PROGRAM MAIN
VAR
    // ── Per-valve motion controllers ──────────────────────────
    fbValve1 : FB_ValveControl;
    fbValve2 : FB_ValveControl;
    fbValve3 : FB_ValveControl;

    // ── NC axis references (linked in TwinCAT I/O mapping) ───
    Axis_Valve1 : AXIS_REF;
    Axis_Valve2 : AXIS_REF;
    Axis_Valve3 : AXIS_REF;

    // ── Infrastructure function blocks ────────────────────────
    fbCsvLogger   : FB_CsvLogger;
    fbMqttManager : FB_MqttManager;

    // ── Internal buffers for MQTT status publishing ───────────
    arrValveSetpoint : ARRAY[1..3] OF REAL;
    arrValveActual   : ARRAY[1..3] OF REAL;
    arrValveSource   : ARRAY[1..3] OF STRING(32);

    // ── Internal helpers ──────────────────────────────────────
    arrPrevHmiSetpoint : ARRAY[1..3] OF REAL := [-1.0, -1.0, -1.0];
    iValve : INT;
END_VAR

// ============================================================
// MAIN PROGRAM OVERVIEW (NOVICE GUIDE)
// ------------------------------------------------------------
// This program is the "orchestrator" of the whole irrigation PLC:
// - It reads operator requests from HMI.
// - It reads remote requests from MQTT (if enabled by operator).
// - It decides which source currently controls each valve.
// - It calls each valve motion FB once per PLC cycle.
// - It logs process values to CSV and mirrors status back to HMI.
//
// Execution sequence each PLC cycle:
// 1) Read/limit HMI commands and reset commands
// 2) Handle source arbitration (HMI vs MQTT)
// 3) Run valve FBs (motion execution)
// 4) Run CSV logger
// 5) Update HMI feedback + overall system health flags
// ============================================================

// ------------------------------------------------------------
// 1) Read and sanitize HMI commands
// ------------------------------------------------------------
GVL_System.Valve[1].HMI_Setpoint := LIMIT(0.0, GVL_HMI.HMI_Valve1_Setpoint, 100.0);
GVL_System.Valve[2].HMI_Setpoint := LIMIT(0.0, GVL_HMI.HMI_Valve2_Setpoint, 100.0);
GVL_System.Valve[3].HMI_Setpoint := LIMIT(0.0, GVL_HMI.HMI_Valve3_Setpoint, 100.0);

GVL_System.Valve[1].Reset_Cmd := GVL_HMI.HMI_Valve1_Reset;
GVL_System.Valve[2].Reset_Cmd := GVL_HMI.HMI_Valve2_Reset;
GVL_System.Valve[3].Reset_Cmd := GVL_HMI.HMI_Valve3_Reset;

IF GVL_HMI.HMI_ResetAll THEN
    GVL_System.Valve[1].Reset_Cmd := TRUE;
    GVL_System.Valve[2].Reset_Cmd := TRUE;
    GVL_System.Valve[3].Reset_Cmd := TRUE;
    GVL_HMI.HMI_ResetAll := FALSE;
END_IF

// ------------------------------------------------------------
// 2) HMI/MQTT command source handling
// ------------------------------------------------------------
// Arbitration rule for beginners:
// - By default, first valid source is HMI.
// - If operator changes HMI setpoint, active source becomes HMI.
// - If a new valid MQTT command arrives and MQTT is enabled,
//   active source changes to MQTT for that valve.
// - Source is stored in GVL_System.Valve[i].Source and shown on HMI.
FOR iValve := 1 TO 3 DO
    IF GVL_System.Valve[iValve].Source = E_ValveSource.NONE THEN
        GVL_System.Valve[iValve].Source := E_ValveSource.HMI;
        GVL_System.Valve[iValve].Active_Setpoint := GVL_System.Valve[iValve].HMI_Setpoint;
    END_IF

    IF ABS(GVL_System.Valve[iValve].HMI_Setpoint - arrPrevHmiSetpoint[iValve]) > 0.001 THEN
        GVL_System.Valve[iValve].Active_Setpoint := GVL_System.Valve[iValve].HMI_Setpoint;
        GVL_System.Valve[iValve].Source := E_ValveSource.HMI;
        arrPrevHmiSetpoint[iValve] := GVL_System.Valve[iValve].HMI_Setpoint;
    END_IF
END_FOR

// Prepare status arrays before MQTT publish
// (This is done in arrays because FB_MqttManager expects fixed arrays.)
arrValveSetpoint[1] := GVL_System.Valve[1].Active_Setpoint;
arrValveSetpoint[2] := GVL_System.Valve[2].Active_Setpoint;
arrValveSetpoint[3] := GVL_System.Valve[3].Active_Setpoint;
arrValveActual[1] := GVL_System.Valve[1].Actual_Position;
arrValveActual[2] := GVL_System.Valve[2].Actual_Position;
arrValveActual[3] := GVL_System.Valve[3].Actual_Position;
arrValveSource[1] := TO_STRING(GVL_System.Valve[1].Source);
arrValveSource[2] := TO_STRING(GVL_System.Valve[2].Source);
arrValveSource[3] := TO_STRING(GVL_System.Valve[3].Source);

// MQTT enable is operator-controlled from HMI checkbox.
// Broker/topic/timing configuration stays fixed in code constants
// (single source of truth = GVL_Config.MQTT_CONFIG).
fbMqttManager(
    bEnable              := GVL_HMI.HMI_MQTT_bEnable,
    stConfig             := GVL_Config.MQTT_CONFIG,
    bApplyConfig         := FALSE,
    bPublish             := GVL_HMI.HMI_MQTT_mPublish,
    sPubTopic            := GVL_Config.MQTT_CONFIG.sMainTopic,
    sPubPayload          := '',
    bSubscribe           := GVL_HMI.HMI_MQTT_bEnable,
    sSubTopic            := GVL_Config.MQTT_CONFIG.SubscribeTopic,
    bUnsubscribe         := FALSE,
    sUnsubTopic          := '',
    bEnableStatusPublish := GVL_HMI.HMI_MQTT_bEnable,
    tStatusPublishTime   := GVL_Config.MQTT_CONFIG.tPublishInterval,
    sStatusTopic         := GVL_Config.MQTT_CONFIG.sMainTopic,
    rValveSetpoint       := arrValveSetpoint,
    rValveActual         := arrValveActual,
    sValveSource         := arrValveSource,
    rTemperature_C       := INT_TO_REAL(GVL_IO.AI_Tmp_1),
    rWaterLevel_Percent  := INT_TO_REAL(GVL_IO.AI_L1V11),
    sTimestamp           := DT_TO_STRING(CURRENT_DT())
);

IF fbMqttManager.bNewRemoteCommand AND GVL_HMI.HMI_MQTT_bEnable THEN
    FOR iValve := 1 TO 3 DO
        GVL_System.Valve[iValve].MQTT_Setpoint   := fbMqttManager.rMqttValveSetpoint[iValve];
        GVL_System.Valve[iValve].Active_Setpoint := GVL_System.Valve[iValve].MQTT_Setpoint;
        GVL_System.Valve[iValve].Source          := E_ValveSource.MQTT;
    END_FOR
END_IF

// ------------------------------------------------------------
// 3) Valve motion control calls (one FB per valve axis)
// Each FB handles homing, move, halt, reset, and fault state machine
// for its own NC axis. MAIN only forwards commands/parameters.
// ------------------------------------------------------------
fbValve1(
    Axis            := Axis_Valve1,
    HMI_Setpoint    := GVL_System.Valve[1].HMI_Setpoint,
    MQTT_Setpoint   := GVL_System.Valve[1].MQTT_Setpoint,
    MQTT_Enabled    := GVL_HMI.HMI_MQTT_bEnable,
    Enable          := TRUE,
    eHomingSelection:= MC_Direct,
    Reset           := GVL_System.Valve[1].Reset_Cmd,
    MoveVelocity    := GVL_Config.VALVE_MOVE_VELOCITY,
    MoveAccel       := GVL_Config.VALVE_MOVE_ACCELERATION,
    MoveDecel       := GVL_Config.VALVE_MOVE_DECELERATION,
    MoveJerk        := GVL_Config.VALVE_MOVE_JERK,
    HomeVelocity    := GVL_Config.VALVE_HOMING_VELOCITY,
    FullStroke_mm   := GVL_Config.VALVE_FULL_STROKE_MM,
    PosTolerance    := GVL_Config.VALVE_POSITION_TOLERANCE,
    Move_Stop       := GVL_HMI.HMI_Valve1_Stop,
    UPDATE          := GVL_HMI.HMI_UPDATE,
    ZeroPosition    := GVL_IO.bBottom_position_1,
    bHoming         := GVL_HMI.HMI_Valve1_Homing,
    Actual_Position => GVL_System.Valve[1].Actual_Position,
    State           => GVL_System.Valve[1].State,
    Source          => GVL_System.Valve[1].Source,
    IsHomed         => GVL_System.Valve[1].IsHomed,
    InPosition      => GVL_System.Valve[1].InPosition,
    IsFault         => GVL_System.Valve[1].IsFault,
    FaultCode       => GVL_System.Valve[1].FaultCode,
    rTarget_mm      => GVL_HMI.Raw_Valve1_Setpoint,
    rActual_mm      => GVL_HMI.Raw_Valve1_Position
);

fbValve2(
    Axis            := Axis_Valve2,
    HMI_Setpoint    := GVL_System.Valve[2].HMI_Setpoint,
    MQTT_Setpoint   := GVL_System.Valve[2].MQTT_Setpoint,
    MQTT_Enabled    := GVL_HMI.HMI_MQTT_bEnable,
    Enable          := TRUE,
    eHomingSelection:= MC_Direct,
    Reset           := GVL_System.Valve[2].Reset_Cmd,
    MoveVelocity    := GVL_Config.VALVE_MOVE_VELOCITY,
    MoveAccel       := GVL_Config.VALVE_MOVE_ACCELERATION,
    MoveDecel       := GVL_Config.VALVE_MOVE_DECELERATION,
    MoveJerk        := GVL_Config.VALVE_MOVE_JERK,
    HomeVelocity    := GVL_Config.VALVE_HOMING_VELOCITY,
    FullStroke_mm   := GVL_Config.VALVE_FULL_STROKE_MM,
    PosTolerance    := GVL_Config.VALVE_POSITION_TOLERANCE,
    Move_Stop       := GVL_HMI.HMI_Valve2_Stop,
    UPDATE          := GVL_HMI.HMI_UPDATE,
    bHoming         := GVL_HMI.HMI_Valve2_Homing,
    Actual_Position => GVL_System.Valve[2].Actual_Position,
    State           => GVL_System.Valve[2].State,
    Source          => GVL_System.Valve[2].Source,
    IsHomed         => GVL_System.Valve[2].IsHomed,
    InPosition      => GVL_System.Valve[2].InPosition,
    IsFault         => GVL_System.Valve[2].IsFault,
    FaultCode       => GVL_System.Valve[2].FaultCode,
    rTarget_mm      => GVL_HMI.Raw_Valve2_Setpoint,
    rActual_mm      => GVL_HMI.Raw_Valve2_Position
);

fbValve3(
    Axis            := Axis_Valve3,
    HMI_Setpoint    := GVL_System.Valve[3].HMI_Setpoint,
    MQTT_Setpoint   := GVL_System.Valve[3].MQTT_Setpoint,
    MQTT_Enabled    := GVL_HMI.HMI_MQTT_bEnable,
    Enable          := TRUE,
    eHomingSelection:= MC_Direct,
    Reset           := GVL_System.Valve[3].Reset_Cmd,
    MoveVelocity    := GVL_Config.VALVE_MOVE_VELOCITY,
    MoveAccel       := GVL_Config.VALVE_MOVE_ACCELERATION,
    MoveDecel       := GVL_Config.VALVE_MOVE_DECELERATION,
    MoveJerk        := GVL_Config.VALVE_MOVE_JERK,
    HomeVelocity    := GVL_Config.VALVE_HOMING_VELOCITY,
    FullStroke_mm   := GVL_Config.VALVE_FULL_STROKE_MM,
    PosTolerance    := GVL_Config.VALVE_POSITION_TOLERANCE,
    Move_Stop       := GVL_HMI.HMI_Valve3_Stop,
    UPDATE          := GVL_HMI.HMI_UPDATE,
    bHoming         := GVL_HMI.HMI_Valve3_Homing,
    Actual_Position => GVL_System.Valve[3].Actual_Position,
    State           => GVL_System.Valve[3].State,
    Source          => GVL_System.Valve[3].Source,
    IsHomed         => GVL_System.Valve[3].IsHomed,
    InPosition      => GVL_System.Valve[3].InPosition,
    IsFault         => GVL_System.Valve[3].IsFault,
    FaultCode       => GVL_System.Valve[3].FaultCode,
    rTarget_mm      => GVL_HMI.Raw_Valve3_Setpoint,
    rActual_mm      => GVL_HMI.Raw_Valve3_Position
);

// ------------------------------------------------------------
// 4) CSV logger
// Logger runs non-blocking state machine and appends one row
// with valve + sensor data when interval/trigger condition is met.
// ------------------------------------------------------------
fbCsvLogger(
    bEnable             := TRUE,
    bForceWrite         := GVL_HMI.WriteTrigger,
    tLogInterval        := GVL_Config.CSV_LOG_INTERVAL_S,
    sBasePath           := GVL_Config.CSV_FILE_PATH,
    sPrefix             := GVL_Config.CSV_FILENAME_PREFIX,
    stValve             := GVL_System.Valve,
    rWaterLevel_Percent := INT_TO_REAL(GVL_IO.AI_L1V11),
    rTemperature_C      := INT_TO_REAL(GVL_IO.AI_Tmp_1),
    dtLastWrite         => GVL_System.CSV_LastWriteTime,
    bError              => GVL_System.CSV_FileError,
    sCurrentFilename    => GVL_System.CSV_CurrentFile,
    eState              => GVL_System.CSV_LoggerState
);

// ------------------------------------------------------------
// 5) Housekeeping and HMI feedback
// Reset one-shot command bits and copy runtime values to display variables.
// ------------------------------------------------------------
GVL_System.Valve[1].Reset_Cmd := FALSE;
GVL_HMI.HMI_Valve1_Reset      := FALSE;
GVL_System.Valve[2].Reset_Cmd := FALSE;
GVL_HMI.HMI_Valve2_Reset      := FALSE;
GVL_System.Valve[3].Reset_Cmd := FALSE;
GVL_HMI.HMI_Valve3_Reset      := FALSE;

GVL_HMI.ACT_Valve1_Position  := GVL_System.Valve[1].Actual_Position;
GVL_HMI.ACT_Valve1_State     := GVL_System.Valve[1].State;
GVL_HMI.ACT_Valve1_Source    := GVL_System.Valve[1].Source;
GVL_HMI.ACT_Valve1_Fault     := GVL_System.Valve[1].IsFault;
GVL_HMI.ACT_Valve1_FaultCode := GVL_System.Valve[1].FaultCode;

GVL_HMI.ACT_Valve2_Position  := GVL_System.Valve[2].Actual_Position;
GVL_HMI.ACT_Valve2_State     := GVL_System.Valve[2].State;
GVL_HMI.ACT_Valve2_Source    := GVL_System.Valve[2].Source;
GVL_HMI.ACT_Valve2_Fault     := GVL_System.Valve[2].IsFault;
GVL_HMI.ACT_Valve2_FaultCode := GVL_System.Valve[2].FaultCode;

GVL_HMI.ACT_Valve3_Position  := GVL_System.Valve[3].Actual_Position;
GVL_HMI.ACT_Valve3_State     := GVL_System.Valve[3].State;
GVL_HMI.ACT_Valve3_Source    := GVL_System.Valve[3].Source;
GVL_HMI.ACT_Valve3_Fault     := GVL_System.Valve[3].IsFault;
GVL_HMI.ACT_Valve3_FaultCode := GVL_System.Valve[3].FaultCode;

GVL_System.AnyFaultActive :=
    GVL_System.Valve[1].IsFault OR
    GVL_System.Valve[2].IsFault OR
    GVL_System.Valve[3].IsFault;

GVL_System.SystemReady :=
    GVL_System.Valve[1].IsHomed AND
    GVL_System.Valve[2].IsHomed AND
    GVL_System.Valve[3].IsHomed AND
    NOT GVL_System.AnyFaultActive;

GVL_HMI.ACT_SystemReady := GVL_System.SystemReady;

END_PROGRAM

(* stored: Version 1.1.0.1, ProductVersion 3.1.4026.18
   POU MAIN: Id {a0f99a09-eccb-42d8-b9bd-167b13d45a91}, SpecialFunc None *)
